{attribute 'linkalways'} 
{attribute 'no_explicit_call' := 'This FB is a CLASS and must be accessed using methods or properties'}
{attribute 'enable_dynamic_creation'}
FUNCTION_BLOCK Node_F_VN_BitwiseAndContainers EXTENDS VisionNode
VAR
    ipSrcContainer1 : _ITcVnContainer;
    ipSrcContainer2 : _ITcVnContainer;
    ipDestContainer : _ITcVnContainer;
    hrPrev : _HRESULT(S_OK);
    hresult : _HRESULT(S_OK);
END_VAR

METHOD PUBLIC  Clone : I_Node
VAR
    pNode : POINTER TO Node_F_VN_BitwiseAndContainers;
END_VAR
pNode := __NEW(Node_F_VN_BitwiseAndContainers);
Clone := pNode^;
END_METHOD

METHOD FB_init : BOOL
VAR_INPUT
    bInitRetains : BOOL; // if TRUE, the retain variables are initialized (warm start / cold start)
    bInCopyCode : BOOL;  // if TRUE, the instance afterwards gets moved into the copy code (online change)
END_VAR
AddInput('ipSrcContainer1', ipSrcContainer1);
AddInput('ipSrcContainer2', ipSrcContainer2);
AddInput('hrPrev', hrPrev);
AddOutput('ipDestContainer', ipDestContainer);
AddOutput('hresult',hresult);
END_METHOD

METHOD PROTECTED OnExecute
hresult.Value := F_VN_BitwiseAndContainers(
    ipSrcContainer1 := ipSrcContainer1.Value,
    ipSrcContainer2 := ipSrcContainer2.Value,
    ipDestContainer := ipDestContainer.Value,
    hrPrev:= hrPrev.Value);
END_METHOD

METHOD PUBLIC PreExecutionCheck
VAR_INPUT
    Check : I_PreExecutionChecks;
END_VAR
Check.IsTrue(ipSrcContainer1.IsValid, 'ipSrcContainer1 must be a valid container');
Check.IsTrue(ipSrcContainer2.IsValid, 'ipSrcContainer2 must be a valid container');
Check.IsTrue(ContainersHaveMatchingTypes(ipSrcContainer1.Value, ipSrcContainer2.Value), 'Source containers must have matching types');
Check.IsTrue(ContainersHaveMatchingNumberOfElements(ipSrcContainer1.Value, ipSrcContainer2.Value), 'Source containers must contain the same number of elements');


//TODO Need to check that container has integer values only.
// SINT, USINT, INT, UINT, DINT, UDINT, ULINT only?
END_METHOD

END_FUNCTION_BLOCK

(* stored: Version 1.1.0.1, ProductVersion 3.1.4024.15
   POU Node_F_VN_BitwiseAndContainers: Id {d9f0532c-af1c-00f5-3d03-786c0fd5f95d}, SpecialFunc None
   Folder Constructor: Id {9447db24-edb6-0597-30a9-04d93bf971b9}
   Method Clone: Id {bafa91a0-e5f0-03a5-38b6-a1f78395b3ee}
   Method FB_init: Id {d6623197-b273-00b6-1803-5474877600b2}
   Method OnExecute: Id {96c2bb51-8cfa-00f9-1f1b-4d350f05e085}
   Method PreExecutionCheck: Id {c16c85df-5503-08b9-0fd3-d5b8647ea019} *)
